(* PLC project  *)

CONFIGURATION CANopen_Manager_SoftMotion
END_CONFIGURATION
